FUNCTION_BLOCK FB_ApplicationMover IMPLEMENTS I_MoverApplication
VAR
	ipMoverStandard	: I_XPlanarMoverStandard;
	
	stProductData	: ST_ProductData;
	eMoverType 		: ST_EMoverLoadType;
	
	nMoverIndex		: INT;
	sMoverID 		: STRING(13) := '00001111';
	
	nTrackId		: UDINT;
	
	// customer Data
	bIsLoaded		: BOOL;	
	stControlData	:ST_ControlData;
	stMoverConfiguration: ST_MoverConfiguration;
	stProcessTask: St_ProcessTask;
	nCurrentStation	: UINT;
	bEnable			: BOOL;
	bError			: BOOL;
	nErrorID		: INT;
	stPartTracking	: ST_PartTrackingData;
	rTrackPos		: LREAL;



END_VAR

METHOD Cycle


VAR_INST
	nTestCounter	: UINT;
	index: UDINT;
	
END_VAR
IF std <> 0 THEN

    std.cycle();

    IF communication.RunAplicationComm THEN 
        FOR index := 1 TO GVL.gc_nMaxNumberMovers DO 

            IF communication.g_Com_Movers[index].IN.id = THIS^.P_MoverID THEN 

                //================= OUT =================

                Communication.g_Com_Movers[index].OUT.Avaiable := (THIS^.std.P_State = 3); // Avaiable

                Communication.g_Com_Movers[index].OUT.Error := THIS^.P_Error; // Error

                Communication.g_Com_Movers[index].OUT.CurrentTaskFinished := stProcessTask.CurrentTaskFinished; // CurrentTaskFinished

                stControlData.StatusWord := THIS^.std.P_State;
                Communication.g_Com_Movers[index].OUT.Status_Word := stControlData.StatusWord; // Status_Word

                Communication.g_Com_Movers[index].OUT.Error_ID := THIS^.P_ErrorID; // Error_ID

                communication.g_Com_Movers[index].out.MoverType := THIS^.stMoverConfiguration.MoverType; // MoverType

                Communication.g_Com_Movers[index].OUT.CurrentStation := THIS^.P_CurrentStation; // CurrentStation

                Communication.g_Com_Movers[index].OUT.LastTask := stProcessTask.LastTask; // LastTask
                Communication.g_Com_Movers[index].OUT.CurrentTask := stProcessTask.CurrentTask; // CurrentTask

                Communication.g_Com_Movers[index].OUT.TrackID := THIS^.P_TrackId; // TrackID

                Communication.g_Com_Movers[index].OUT.TrackPos := THIS^.P_TrackPos; // TrackPos

                Communication.g_Com_Movers[index].OUT.Id := THIS^.P_MoverID; // Id

                Communication.g_Com_Movers[index].OUT.position.vec := THIS^.std.P_ActPosition;
                Communication.g_Com_Movers[index].OUT.Position.vec.x := THIS^.std.P_ActPosition.x;
                Communication.g_Com_Movers[index].OUT.Position.vec.y := THIS^.std.P_ActPosition.y;
                Communication.g_Com_Movers[index].OUT.Position.vec.c := THIS^.std.P_ActPosition.c; // Position

                Communication.g_Com_Movers[index].OUT.PartTracking := THIS^.P_PartTracking; // Part tracking

                //================= IN =================

                THIS^.P_Enable := Communication.g_Com_Movers[index].IN.Enable; // Enable

                IF Communication.g_Com_Movers[index].IN.Reset THEN
                    ipMoverStandard.Reset(slogMessage := 'mover reset');
                END_IF // Reset

                stMoverConfiguration.MoverType := Communication.g_Com_Movers[index].IN.MoverType;
                IF communication.g_Com_Movers[index].IN.MoverType = 1 THEN 
                    eMoverType := ST_EMoverLoadType.Wellplate;
                ELSIF communication.g_Com_Movers[index].IN.MoverType = 2 THEN 
                    eMoverType := ST_EMoverLoadType.Gripper;
                ELSIF communication.g_Com_Movers[index].IN.MoverType = 3 THEN 
                    eMoverType := ST_EMoverLoadType.PipetteTips;
                END_IF	// Mover Type

                stControlData.ControlWord := communication.g_Com_Movers[index].IN.ControlWord; // ControlWord

                stProcessTask.TaskToProcessed := Communication.g_Com_Movers[index].IN.TaskToProcessed; // TaskToProcced

                // ID — użyte wyżej do dopasowania slotu

                stMoverConfiguration.WellplateData := Communication.g_Com_Movers[index].IN.WellplateData; // WellplateData

            END_IF
        END_FOR
    END_IF

END_IF
END_METHOD

METHOD ManualMovement : BOOL
VAR_INPUT
	bReset: bool;
END_VAR

VAR_INST
	nTestCounter	: UINT;
	index: UDINT;
	Com_Index: UDINT;
	nMovementSequence : UDINT;
	
	
END_VAR

VAR
	ManMovements: 	ST_ManualMovements;
	targetPos 						:  PositionXYC;
	fTargetPosOnTrack 				: LREAL;
	stOptionsJoinTrack				: ST_JoinTrackOptions;
	stMoveOnTrackOptions			: ST_MoveOnTrackOptions;
	stMoveToPositionOptions			: ST_MoveToPositionOptions;
	bMoversJoined 					: BOOL;
	bMoverError						: BOOL;
	bMoversInPos					: BOOL;
	strInfo							: STRING;
	
END_VAR
	IF communication.RunAplicationComm THEN 
		FOR index:=1 TO GVL.gc_nMaxNumberMovers DO 
			
			IF communication.g_Com_Movers[index].IN.id= THIS^.P_MoverID THEN
				
				ManMovements:= communication.g_Com_Movers[index].ManualMovements;
				Com_Index:=index;
				
			END_IF
			
		END_FOR
		
	END_IF
	
	
	
	IF bReset OR  Communication.g_Com_GlobalState.IN.Stop   OR Communication.g_Com_GlobalState.IN.Reset THEN 
	ManualMovement := FALSE;
	nMovementSequence := 0;
END_IF

CASE nMovementSequence OF
	

0: //init
		
 	// wait for enabling  process 
			 IF Communication.g_Com_GlobalState.IN.Start AND NOT Communication.g_Com_GlobalState.IN.EOC_Stop  AND Com_Index <>0 THEN 
				IF Communication.g_Com_GlobalState.IN.ProgramType =2 THEN 
					  nMovementSequence := 100;
				
					   ELSIF Communication.g_Com_GlobalState.IN.ProgramType =3 THEN 
					  nMovementSequence := 200;
				END_IF								
					 
			 END_IF
			 




100:	 // position test 
	
		// leave track
		IF ipMoverStandard.P_CommandMode= MC_PLANAR_MOVER_COMMAND_MODE.OnTrack AND  NOT ipMoverStandard.P_Busy THEN

			ipMoverStandard.LeaveTrackInPosition( strInfo, FALSE);
			nMovementSequence := nMovementSequence +1;
		ELSE 
			nMovementSequence := 110;
		END_IF


101:
			IF ipMoverStandard.P_LeaveTrackInPosition.Done THEN
				P_TrackId:=0;
				nMovementSequence := 110;
			ELSIF ipMoverStandard.P_LeaveTrackInPosition.Error THEN
				nMovementSequence := nMovementSequence +4;
			END_IF	
				


110://setup state 
		IF NOT ManMovements.FreeMove.move_position_CMD_enable THEN 
				ManMovements.FreeMove.move_position_CMD_done:= FALSE;
				communication.g_Com_Movers[Com_Index].ManualMovements:=ManMovements;
		END_IF
						nMovementSequence := nMovementSequence +  1;					  
				
111: 	//execute command 
stMoveToPositionOptions.useOrientation:= TRUE;
	targetPos.x:=	ManMovements.FreeMove.move_position.x ;
	targetPos.y:=	ManMovements.FreeMove.move_position.y;
	targetPos.C:=	ManMovements.FreeMove.move_position.C;
					 // targetpos.ShiftByXy(ManMovements.move_position.x,ManMovements.move_position.y);
				
	


			IF  ManMovements.FreeMove.move_position_CMD_enable AND NOT ManMovements.FreeMove.move_position_CMD_done  THEN 
					ipMoverStandard.MoveToPositionEXt('move to XY', targetPos, 100, 2500, 2500, 25000,stMoveToPositionOptions);
					nMovementSequence := nMovementSequence +  1;
			ELSE
				nMovementSequence := 0;
			END_IF
				
		
	
	
112: 	// check commad result 

		
		IF ipMoverStandard.P_MoveToPositionExt.Done THEN
			ManMovements.FreeMove.move_position_CMD_done:= TRUE;
			communication.g_Com_Movers[Com_Index].ManualMovements:=ManMovements;
			nMovementSequence :=  0;
		ELSIF ipMoverStandard.P_MoveToPositionExt.Error THEN
			nMovementSequence := nMovementSequence +  3;
		END_IF				
		
		
200:
		 IF NOT ManMovements.MoveTrack.move_track_CMD_done THEN 
				IF ManMovements.MoveTrack.join_track AND ManMovements.MoveTrack.move_track_no<>0 THEN 
					nMovementSequence := 210;
				ELSIF ManMovements.MoveTrack.leave_track THEN
					nMovementSequence := 220;
				ELSIF ManMovements.MoveTrack.move_track AND ManMovements.MoveTrack.move_track_no<>0 THEN 
					nMovementSequence := 230;
				ELSE
					nMovementSequence := 0;
				END_IF
		END_IF
		
		IF NOT ManMovements.MoveTrack.move_track_CMD_enable THEN 
			ManMovements.MoveTrack.move_track_CMD_done := FALSE;
			communication.g_Com_Movers[Com_Index].ManualMovements:=ManMovements;
		END_IF

210:	
		stOptionsJoinTrack.useOrientation := TRUE;
	
		IF (ipMoverStandard.P_CommandMode<> MC_PLANAR_MOVER_COMMAND_MODE.OnTrack OR  INT_TO_UDINT(ManMovements.MoveTrack.move_track_no)<>P_TrackId)
			AND NOT ipMoverStandard.P_Busy
			AND ManMovements.MoveTrack.move_track_CMD_enable THEN
			ipMoverStandard.JoinTrack('Joining track', GVL.g_Tracks[ManMovements.MoveTrack.move_track_no].std, 250, 1250, 12500, stOptionsJoinTrack);
				nMovementSequence := nMovementSequence + 1;
			ELSE 
				nMovementSequence := 0;
		END_IF
	
	
		
211:
	
			bMoversJoined := ipMoverStandard.P_JoinTrack.Done;
			bMoverError :=  ipMoverStandard.P_JoinTrack.Error;			
		
	IF bMoversJoined THEN
		ManMovements.MoveTrack.move_track_CMD_done:=TRUE;
		communication.g_Com_Movers[Com_Index].ManualMovements:=ManMovements;
		P_TrackId:=INT_TO_UDINT(ManMovements.MoveTrack.move_track_no);
		nMovementSequence := 0;
	ELSIF bMoverError THEN
 			nMovementSequence := nMovementSequence + 4;
	END_IF

		
	
		
220:
		
		IF ipMoverStandard.P_CommandMode= MC_PLANAR_MOVER_COMMAND_MODE.OnTrack AND  NOT ipMoverStandard.P_Busy AND ManMovements.MoveTrack.move_track_CMD_enable  THEN

			ipMoverStandard.LeaveTrackInPosition( strInfo, FALSE);
			nMovementSequence := nMovementSequence +1;
		ELSE 
			nMovementSequence := 0;
		END_IF


221:
			IF ipMoverStandard.P_LeaveTrackInPosition.Done THEN
				ManMovements.MoveTrack.move_track_CMD_done:=TRUE;
				communication.g_Com_Movers[Com_Index].ManualMovements:=ManMovements;
				P_TrackId:=0;
				nMovementSequence := 0;
			ELSIF ipMoverStandard.P_LeaveTrackInPosition.Error THEN
				nMovementSequence := nMovementSequence +4;
			END_IF	
			
230:

		
		stMoveOnTrackOptions.gap := 120;
		fTargetPosOnTrack:=ManMovements.MoveTrack.move_track_position;
		stMoveOnTrackOptions.dynamicMode := MC_DYNAMICS_REDUCTION_MODE.AccelerationLimitedVelocity;
		stMoveOnTrackOptions.direction := MC_DIRECTION.mcDirectionShortestWay;
		IF   NOT ipMoverStandard.P_Busy AND ManMovements.MoveTrack.move_track_CMD_enable  THEN
				 ipMoverStandard.MoveOnTrackEXT('move on track', GVL.g_Tracks[ManMovements.MoveTrack.move_track_no].std, fTargetPosOnTrack,
								300, 3000, 15000, stMoveOnTrackOptions);
				nMovementSequence := nMovementSequence +1;
		 END_IF
		 


	231:
			bMoversInPos :=  ipMoverStandard.P_MoveOnTrackExt.Done;
			bMoverError := ipMoverStandard.P_MoveOnTrackExt.Error;
	
		
		IF bMoversInPos THEN
			ManMovements.MoveTrack.move_track_CMD_done:=TRUE;
			communication.g_Com_Movers[Com_Index].ManualMovements:=ManMovements;
			nMovementSequence := 0;
		ELSIF bMoverError THEN
			nMovementSequence := nMovementSequence +  3;
		END_IF
			
			
			
	END_CASE
END_METHOD

PROPERTY P_ControlData : Reference to ST_ControlData
GET
P_ControlData := stControlData;
END_GET
SET
stControlData := P_ControlData;
END_SET
END_PROPERTY

PROPERTY P_CurrentStation : UINT
GET
P_CurrentStation := nCurrentStation;
END_GET
SET
nCurrentStation := P_CurrentStation;
END_SET
END_PROPERTY

PROPERTY P_Enable : BOOL
GET
P_Enable := bEnable;
END_GET
SET
bEnable := P_Enable;
END_SET
END_PROPERTY

PROPERTY P_Error : BOOL
GET
P_Error := bError;
END_GET
SET
bError := P_Error;
END_SET
END_PROPERTY

PROPERTY P_ErrorID : INT
GET
P_ErrorID := nErrorID;
END_GET
SET
nErrorID := P_ErrorID;
END_SET
END_PROPERTY

PROPERTY P_MoverConfiguration : Reference to  ST_MoverConfiguration
GET
P_MoverConfiguration := stMoverConfiguration;
END_GET
SET
stMoverConfiguration := P_MoverConfiguration;
END_SET
END_PROPERTY

PROPERTY P_MoverID : STRING
GET
P_MoverID := sMoverID;
END_GET
SET
sMoverID := P_MoverID;
END_SET
END_PROPERTY

PROPERTY P_MoverIndex : INT
GET
P_MoverIndex := nMoverIndex;
END_GET
SET
nMoverIndex := P_MoverIndex;
END_SET
END_PROPERTY

PROPERTY P_PartTracking : ST_PartTrackingData
GET
P_PartTracking := stPartTracking;
END_GET
SET
stPartTracking := P_PartTracking;
END_SET
END_PROPERTY

PROPERTY P_ProcessTask : ST_ProcessTask
GET
P_ProcessTask := stProcessTask;
END_GET
SET
stProcessTask := P_ProcessTask;
END_SET
END_PROPERTY

PROPERTY P_ProductData : Reference to ST_ProductData
GET
P_ProductData REF= stProductData;
END_GET
SET
stProductData := P_ProductData;
END_SET
END_PROPERTY

PROPERTY P_TrackId : UDINT
GET
P_TrackId := nTrackId;
END_GET
SET
nTrackId := P_TrackId;
END_SET
END_PROPERTY

PROPERTY P_TrackPos : LREAL
GET
P_TrackPos := rTrackPos;
END_GET
SET
rTrackPos := P_TrackPos;
END_SET
END_PROPERTY

PROPERTY std : I_XPlanarMoverStandard
GET
IF ipMoverStandard <> 0 THEN
	std := ipMoverStandard;	
END_IF
END_GET
SET
ipMoverStandard := std;
END_SET
END_PROPERTY

END_FUNCTION_BLOCK

(* stored: Version 1.1.0.1
   POU FB_ApplicationMover: Id {40b5c66d-1fb4-4d55-9f96-3f23301af31f}, SpecialFunc None
   Method Cycle: Id {3db1001d-9da7-43c7-a358-11235832af95}
   Method ManualMovement: Id {7865894f-0036-4baf-a267-0db1d28c8243}
   Property P_ControlData: Id {2455e71b-fb83-4044-b907-3e616e6c3fda}
   Get Get: Id {9b17cc24-af14-47f7-bb6d-635fc676933d}
   Set Set: Id {9340ef7c-3967-4a37-992a-4da9010b0d18}
   Property P_CurrentStation: Id {bdf8ca0a-4b3c-4c2f-8aac-7cbbcd93f7f8}
   Get Get: Id {92508fd3-51a5-4c1f-9f0b-2df485289604}
   Set Set: Id {47498548-63c6-4774-a55f-4ef95acf0df9}
   Property P_Enable: Id {480778eb-b003-4670-840a-8fb13ad83e25}
   Get Get: Id {13960bad-1de1-488e-b02c-4369e0714316}
   Set Set: Id {e618bda7-7fc1-4950-ad2d-05fdd9b1fd5e}
   Property P_Error: Id {02316ece-80a4-46a7-8c3b-9eac5fa8a56f}
   Get Get: Id {d336fe54-7c55-4225-9cd4-6cb06492095e}
   Set Set: Id {d885d4c1-389a-4bae-b760-e1ceca4ff91c}
   Property P_ErrorID: Id {516692b1-d5c8-4382-a043-b8aca770e5b4}
   Get Get: Id {a3de3b84-3b63-4208-b092-b8bdc33e2307}
   Set Set: Id {d05e65a1-e21f-4a39-83d3-8c43c4779a21}
   Property P_MoverConfiguration: Id {cfe16262-f9ee-41e2-9e7e-647c990c55f5}
   Get Get: Id {75c82f30-bcc9-4d22-bae8-67a779aac687}
   Set Set: Id {e3a6a65f-4430-4204-90e3-609c1eb17e7e}
   Property P_MoverID: Id {ceaf460d-d28b-4605-a088-d68a1efdefde}
   Get Get: Id {246c1b7c-a7c3-415e-a7a1-5fdd75505ec4}
   Set Set: Id {a48c6801-c6b0-48e8-befc-74830e92c1cc}
   Property P_MoverIndex: Id {8b0bebb8-d22b-43e1-ab25-8038159fc710}
   Get Get: Id {6f9fc754-362d-4beb-b50e-e77684f8d50a}
   Set Set: Id {e9f36281-f830-4039-8a28-5be43aca55c3}
   Property P_PartTracking: Id {ae2fd539-833e-4434-bde9-099977f3ec3e}
   Get Get: Id {0d17c951-4c1e-4717-a139-0925ffcf3b89}
   Set Set: Id {d22c3268-5f7d-460a-9db2-6e4bc9467b84}
   Property P_ProcessTask: Id {15a1423a-be1f-4d14-88f2-a95cd229bed9}
   Get Get: Id {7bdaac9d-2cac-4616-96a6-38473a7bb3f5}
   Set Set: Id {0c0cce35-0525-420c-b754-e161c1a641f3}
   Property P_ProductData: Id {2fbfbc33-cad6-4c1a-b194-3c225a2cf1a2}
   Get Get: Id {4bf4c121-923d-40dd-9c53-7ec22e020235}
   Set Set: Id {d33adc77-a2c9-4f4a-8e6a-c148905050cb}
   Property P_TrackId: Id {bb3a46f6-fd72-439f-b5bc-ae327bc94714}
   Get Get: Id {46b8b84e-3f2c-4789-b5d6-57d0e1a81c42}
   Set Set: Id {d5f18ced-3aa1-4f6f-8451-8cfd636c29e7}
   Property P_TrackPos: Id {1214d7e0-0cd1-4fec-8e94-8c28efb822da}
   Get Get: Id {9bb892b7-7e79-46e0-ad0b-108e3303635a}
   Set Set: Id {f141e5bc-486e-4472-b936-03e94861a68b}
   Property std: Id {74c2e056-88c5-47b5-acb8-9968b5751165}
   Get Get: Id {fdfe9a14-b3ed-40dd-b13f-11a53d96eb71}
   Set Set: Id {75695d29-ba0d-4136-a3f2-f10c3a65b76b} *)
